# EPICS substitutions: icefrdgeSup/loop.substitutions
file loop.template {
  pattern
    {P, PORT, LOOP_NUM}

    {"\$(P)", "\$(PORT)", "1"}
    {"\$(P)", "\$(PORT)", "2"}
}
